FUNCTION MA_Jog : INT

VAR_INPUT
	Speed: REAL:=0;
END_VAR


VAR_IN_OUT
	Axis: Motion_Axis;
END_VAR

VAR
	i: INT:=0;
END_VAR

Axis.IN_Closed_Open_Loop:=0;
Axis.IN_Enable_Control:=1;
Axis.OL_IN_Analog:=Speed;
Axis.OL_IN_Slave_Enable:=0;
Axis.OL_Move_Type:=0;
Axis.OL_IN_Bump_Duration:= T#0MS;  //Timer for Bump Type of Move
Axis.OL_IN_Bump_Trigger:= 0;

END_FUNCTION

(* stored: Version 1.1.0.1, ProductVersion 3.1.4020.12
   POU MA_Jog: Id {e9167776-839b-4403-a452-9c67db02f538}, SpecialFunc None *)
